{attribute 'GeneratedUsingTerminal: EK1100-0000-0018'}
{attribute addProperty BoxType "EK1100-0000-0018"}
{attribute addProperty Id "Beckhoff_EPP1xxxEK1122Beckhoff_EPP1xxxEK1122_5ECABF39762"}
{attribute addProperty CRC "844117325"}
{attribute addProperty Size "762"}
TYPE Beckhoff_EPP1xxx_3250354D EXTENDS EK1100_1FC0878B :
STRUCT
	{attribute addProperty Name "Beckhoff EPP1xxxEK1122"}
	{attribute addProperty PreviousPort "Beckhoff EPP1xxx : B"}
	Beckhoff_EPP1xxxEK1122 : Beckhoff_EPP1xxxEK1122_5ECABF39;
END_STRUCT
END_TYPE

(* stored: Version 1.2.0.0, ProductVersion 3.1.4024.11
   DUT Beckhoff_EPP1xxx_3250354D: Id {9e8d860f-fc30-439e-9be1-45f797b7166e} *)
